(* IEC 61131-3 sources: teller/JD_Teller_LC2_V11/Class/Visu_Boxediter_MinMax, 1 file *)

(* ---- Visu_Boxediter_MinMax.st ---- *)
(*!
<Class
	Name               = "Visu_Boxediter_MinMax"
	Revision           = "1.2"
	RealtimeTask       = "false"
	CyclicTask         = "false"
	BackgroundTask     = "false"
	Sigmatek           = "false"
	OSInterface        = "false"
	HighPriority       = "false"
	Automatic          = "false"
	UpdateMode         = "Prescan"
	SharedCommandTable = "true"
	Objectsize         = "(750,1320)">
	<Channels>
		<Server Name="ClassSvr" Visualized="false" Initialize="false" WriteProtected="true" Retentive="false"/>
		<Server Name="s_BoxMogelijkopMachine" Visualized="true" Initialize="false" WriteProtected="false" Retentive="false"/>
		<Server Name="s_BoxType" Visualized="true" Initialize="false" WriteProtected="false" Retentive="false"/>
		<Server Name="s_Doosnaam" Visualized="true" Initialize="false" WriteProtected="true" Retentive="false"/>
		<Server Name="s_MaxLength" Visualized="true" Initialize="false" WriteProtected="false" Retentive="false"/>
		<Server Name="s_MaxWidth" Visualized="true" Initialize="false" WriteProtected="false" Retentive="false"/>
		<Server Name="s_Offset_Max" Visualized="true" Initialize="false" WriteProtected="false" Retentive="false"/>
		<Server Name="s_Offset_Min" Visualized="true" Initialize="false" WriteProtected="false" Retentive="false"/>
		<Server Name="s_Refresh_Values" Visualized="false" Initialize="false" WriteProtected="false" Retentive="false"/>
		<Server Name="s_T_Max" Visualized="true" Initialize="false" WriteProtected="false" Retentive="false"/>
		<Server Name="s_T_Min" Visualized="true" Initialize="false" WriteProtected="false" Retentive="false"/>
		<Server Name="s_U_Max" Visualized="true" Initialize="false" WriteProtected="false" Retentive="false"/>
		<Server Name="s_U_Min" Visualized="true" Initialize="false" WriteProtected="false" Retentive="false"/>
		<Server Name="s_V_Max" Visualized="true" Initialize="false" WriteProtected="false" Retentive="false"/>
		<Server Name="s_V_Min" Visualized="true" Initialize="false" WriteProtected="false" Retentive="false"/>
		<Server Name="s_W_Max" Visualized="true" Initialize="false" WriteProtected="false" Retentive="false"/>
		<Server Name="s_W_Min" Visualized="true" Initialize="false" WriteProtected="false" Retentive="false"/>
		<Server Name="s_X_Max" Visualized="true" Initialize="false" WriteProtected="false" Retentive="false"/>
		<Server Name="s_X_Min" Visualized="true" Initialize="false" WriteProtected="false" Retentive="false"/>
		<Server Name="s_Y_Max" Visualized="true" Initialize="false" WriteProtected="false" Retentive="false"/>
		<Server Name="s_Y_Min" Visualized="true" Initialize="false" WriteProtected="false" Retentive="false"/>
		<Server Name="s_Z_Max" Visualized="true" Initialize="false" WriteProtected="false" Retentive="false"/>
		<Server Name="s_Z_Min" Visualized="true" Initialize="false" WriteProtected="false" Retentive="false"/>
		<Client Name="c_Boxtype" Required="false" Internal="false"/>
		<Client Name="c_DoosData" Required="true" Internal="false"/>
		<Client Name="c_Refresh_Values" Required="true" Internal="false"/>
	</Channels>
	<RevDoku>
		<Owner Company="JD" Author="J van Diggelen"/>
		<Dokumentation Revision="1.2" Date="2014-04-29" Author="J van Diggelen" Company="JD" Description="doos 14 toegevoegd"/>
		<Dokumentation Revision="1.1" Date="2013-09-21" Author="J van Diggelen" Company="JD" Description="input warning opgelost"/>
		<Dokumentation Revision="1.0" Date="2011-12-06" Author="J van Diggelen" Company="JD" Description="De Visuwaarde van de Service settings van de boxeditor"/>
	</RevDoku>
</Class>
*)
Visu_Boxediter_MinMax : CLASS
  //Servers:
	ClassSvr 	: SvrChCmd_DINT;
	s_Doosnaam 	: SvrCh_tDoosnaam;
	s_BoxType 	: SvrCh_DINT;
	s_BoxMogelijkopMachine 	: SvrCh_DINT;
	s_MaxLength 	: SvrCh_DINT;
	s_MaxWidth 	: SvrCh_DINT;
	s_T_Max 	: SvrCh_DINT;
	s_T_Min 	: SvrCh_DINT;
	s_U_Max 	: SvrCh_DINT;
	s_U_Min 	: SvrCh_DINT;
	s_V_Max 	: SvrCh_DINT;
	s_V_Min 	: SvrCh_DINT;
	s_W_Max 	: SvrCh_DINT;
	s_W_Min 	: SvrCh_DINT;
	s_X_Max 	: SvrCh_DINT;
	s_X_Min 	: SvrCh_DINT;
	s_Y_Max 	: SvrCh_DINT;
	s_Y_Min 	: SvrCh_DINT;
	s_Z_Max 	: SvrCh_DINT;
	s_Z_Min 	: SvrCh_DINT;
	s_Offset_Max 	: SvrCh_DINT;
	s_Offset_Min 	: SvrCh_DINT;
	s_Refresh_Values 	: SvrCh_DINT;
  //Clients:
	c_DoosData 	: CltChCmd_RAMex;
	c_Boxtype 	: CltCh_DINT;
	c_Refresh_Values 	: CltCh_DINT;
  //Variables:
		DoosData 	: ^tDoosParameters;
  //Functions:

	FUNCTION VIRTUAL GLOBAL Init;

	FUNCTION VIRTUAL GLOBAL Background
		VAR_INPUT
			EAX 	: UDINT;
		END_VAR
		VAR_OUTPUT
			state (EAX) 	: UDINT;
		END_VAR;

	FUNCTION VIRTUAL GLOBAL s_BoxType::Write
		VAR_INPUT
			input (EAX) 	: DINT;
		END_VAR
		VAR_OUTPUT
			result (EAX) 	: DINT;
		END_VAR;

	FUNCTION VIRTUAL GLOBAL s_BoxMogelijkopMachine::Write
		VAR_INPUT
			input (EAX) 	: DINT;
		END_VAR
		VAR_OUTPUT
			result (EAX) 	: DINT;
		END_VAR;

	FUNCTION VIRTUAL GLOBAL s_MaxLength::Write
		VAR_INPUT
			input (EAX) 	: DINT;
		END_VAR
		VAR_OUTPUT
			result (EAX) 	: DINT;
		END_VAR;

	FUNCTION VIRTUAL GLOBAL s_MaxWidth::Write
		VAR_INPUT
			input (EAX) 	: DINT;
		END_VAR
		VAR_OUTPUT
			result (EAX) 	: DINT;
		END_VAR;

	FUNCTION VIRTUAL GLOBAL s_T_Max::Write
		VAR_INPUT
			input (EAX) 	: DINT;
		END_VAR
		VAR_OUTPUT
			result (EAX) 	: DINT;
		END_VAR;

	FUNCTION VIRTUAL GLOBAL s_T_Min::Write
		VAR_INPUT
			input (EAX) 	: DINT;
		END_VAR
		VAR_OUTPUT
			result (EAX) 	: DINT;
		END_VAR;

	FUNCTION VIRTUAL GLOBAL s_U_Max::Write
		VAR_INPUT
			input (EAX) 	: DINT;
		END_VAR
		VAR_OUTPUT
			result (EAX) 	: DINT;
		END_VAR;

	FUNCTION VIRTUAL GLOBAL s_U_Min::Write
		VAR_INPUT
			input (EAX) 	: DINT;
		END_VAR
		VAR_OUTPUT
			result (EAX) 	: DINT;
		END_VAR;

	FUNCTION VIRTUAL GLOBAL s_V_Max::Write
		VAR_INPUT
			input (EAX) 	: DINT;
		END_VAR
		VAR_OUTPUT
			result (EAX) 	: DINT;
		END_VAR;

	FUNCTION VIRTUAL GLOBAL s_V_Min::Write
		VAR_INPUT
			input (EAX) 	: DINT;
		END_VAR
		VAR_OUTPUT
			result (EAX) 	: DINT;
		END_VAR;

	FUNCTION VIRTUAL GLOBAL s_W_Max::Write
		VAR_INPUT
			input (EAX) 	: DINT;
		END_VAR
		VAR_OUTPUT
			result (EAX) 	: DINT;
		END_VAR;

	FUNCTION VIRTUAL GLOBAL s_W_Min::Write
		VAR_INPUT
			input (EAX) 	: DINT;
		END_VAR
		VAR_OUTPUT
			result (EAX) 	: DINT;
		END_VAR;

	FUNCTION VIRTUAL GLOBAL s_X_Max::Write
		VAR_INPUT
			input (EAX) 	: DINT;
		END_VAR
		VAR_OUTPUT
			result (EAX) 	: DINT;
		END_VAR;

	FUNCTION VIRTUAL GLOBAL s_X_Min::Write
		VAR_INPUT
			input (EAX) 	: DINT;
		END_VAR
		VAR_OUTPUT
			result (EAX) 	: DINT;
		END_VAR;

	FUNCTION VIRTUAL GLOBAL s_Y_Max::Write
		VAR_INPUT
			input (EAX) 	: DINT;
		END_VAR
		VAR_OUTPUT
			result (EAX) 	: DINT;
		END_VAR;

	FUNCTION VIRTUAL GLOBAL s_Y_Min::Write
		VAR_INPUT
			input (EAX) 	: DINT;
		END_VAR
		VAR_OUTPUT
			result (EAX) 	: DINT;
		END_VAR;

	FUNCTION VIRTUAL GLOBAL s_Z_Max::Write
		VAR_INPUT
			input (EAX) 	: DINT;
		END_VAR
		VAR_OUTPUT
			result (EAX) 	: DINT;
		END_VAR;

	FUNCTION VIRTUAL GLOBAL s_Z_Min::Write
		VAR_INPUT
			input (EAX) 	: DINT;
		END_VAR
		VAR_OUTPUT
			result (EAX) 	: DINT;
		END_VAR;

	FUNCTION VIRTUAL GLOBAL s_Offset_Max::Write
		VAR_INPUT
			input (EAX) 	: DINT;
		END_VAR
		VAR_OUTPUT
			result (EAX) 	: DINT;
		END_VAR;

	FUNCTION VIRTUAL GLOBAL s_Offset_Min::Write
		VAR_INPUT
			input (EAX) 	: DINT;
		END_VAR
		VAR_OUTPUT
			result (EAX) 	: DINT;
		END_VAR;

	FUNCTION VIRTUAL GLOBAL s_Refresh_Values::Write
		VAR_INPUT
			input (EAX) 	: DINT;
		END_VAR
		VAR_OUTPUT
			result (EAX) 	: DINT;
		END_VAR;
  //Tables:
	FUNCTION @STD
		VAR_OUTPUT
			ret_code	: CONFSTATES;
		END_VAR;
	FUNCTION GLOBAL TAB @CT_;
END_CLASS;

#pragma usingLtd RAMex

//Er is in de pointer variabele doosdata een array structuur gemaakt om bij elk type doos de minimale en maximale
//waardes in een service scherm te veranderen.

FUNCTION VIRTUAL GLOBAL Visu_Boxediter_MinMax::Init

  if c_DoosData.GetSize() <> sizeof(tDoosParameters) then
     c_DoosData.SetSize(udSize:=sizeof(tDoosParameters));
  end_if;

  if _FirstScan = 1 then

     DoosData := (c_DoosData.GetDataPtr())$^tDoosParameters;
     s_BoxType := c_Boxtype;
     s_BoxType.Write(s_BoxType);

  end_if;

END_FUNCTION

FUNCTION VIRTUAL GLOBAL Visu_Boxediter_MinMax::Background
	VAR_INPUT
		EAX 	: UDINT;
	END_VAR
	VAR_OUTPUT
		state (EAX) 	: UDINT;
	END_VAR

	state := READY;

END_FUNCTION

FUNCTION VIRTUAL GLOBAL Visu_Boxediter_MinMax::s_BoxType::Write
	VAR_INPUT
		input (EAX) 	: DINT;
	END_VAR
	VAR_OUTPUT
		result (EAX) 	: DINT;
	END_VAR

	s_BoxType := input;

  // doostype moet tussen 1 en 14 liggen
  if    s_BoxType <1 then
        s_BoxType :=1;
  elsif s_BoxType >14 then
        s_BoxType :=14;
  end_if;

 	result := s_BoxType;

  //Doostype
  if     s_BoxType = 1 then
         s_Doosnaam := Langsnaad;
  elsif  s_BoxType = 2 then
         s_Doosnaam := Driepunt;
  elsif  s_BoxType = 3 then
         s_Doosnaam := Driepunt_Vakverdeling;
  elsif  s_BoxType = 4 then
         s_Doosnaam := Vierpunt_Infold;
  elsif  s_BoxType = 5 then
         s_Doosnaam := Vierpunt_Outfold;
  elsif  s_BoxType = 6 then
         s_Doosnaam := Vierpunt_Deksel;
  elsif  s_BoxType = 7 then
         s_Doosnaam := Vierpunt_Dubbele_Wand;
  elsif  s_BoxType = 8 then
         s_Doosnaam := Zespunt_In_In;
  elsif  s_BoxType = 9 then
         s_Doosnaam := Zespunt_In_Out;
  elsif  s_BoxType = 10 then
         s_Doosnaam := Zespunt_In_In_Gespiegeld;
  elsif  s_BoxType = 11 then
         s_Doosnaam := Driepunt_Gespiegeld;
  elsif  s_BoxType = 12 then
         s_Doosnaam := Driepunt;
  elsif  s_BoxType = 13 then
         s_Doosnaam := Langsnaad2;
  elsif  s_BoxType = 14 then
         s_Doosnaam := Driepunt2;
  end_if;

  //Serverwaardes schrijven met variabelen voor type doos

  s_MaxLength := DoosData^.MinMax[s_BoxType].Max_Invoer_Lengte;
  s_MaxWidth  := DoosData^.MinMax[s_BoxType].Max_Invoer_Breedte;
  s_BoxMogelijkopMachine := DoosData^.MinMax[s_BoxType].BoxMogelijk;
  s_T_Max     := DoosData^.MinMax[s_BoxType].T_Max;
  s_T_Min     := DoosData^.MinMax[s_BoxType].T_Min;
  s_U_Max     := DoosData^.MinMax[s_BoxType].U_Max;
  s_U_Min     := DoosData^.MinMax[s_BoxType].U_Min;
  s_V_Min     := DoosData^.MinMax[s_BoxType].V_Min;
  s_V_Max     := DoosData^.MinMax[s_BoxType].V_Max;
  s_W_Max     := DoosData^.MinMax[s_BoxType].W_Max;
  s_W_Min     := DoosData^.MinMax[s_BoxType].W_Min;
  s_X_Max     := DoosData^.MinMax[s_BoxType].X_Max;
  s_X_Min     := DoosData^.MinMax[s_BoxType].X_Min;
  s_Y_Max     := DoosData^.MinMax[s_BoxType].Y_Max;
  s_Y_Min     := DoosData^.MinMax[s_BoxType].Y_Min;
  s_Z_Max     := DoosData^.MinMax[s_BoxType].Z_Max;
  s_Z_Min     := DoosData^.MinMax[s_BoxType].Z_Min;
  s_Offset_Max:= DoosData^.MinMax[s_BoxType].Offset_Max;
  s_Offset_Min:= DoosData^.MinMax[s_BoxType].Offset_Min;

END_FUNCTION

FUNCTION VIRTUAL GLOBAL Visu_Boxediter_MinMax::s_BoxMogelijkopMachine::Write
	VAR_INPUT
		input (EAX) 	: DINT;
	END_VAR
	VAR_OUTPUT
		result (EAX) 	: DINT;
	END_VAR

  s_BoxMogelijkopMachine := input;
  DoosData^.MinMax[s_BoxType].BoxMogelijk := to_bool(s_BoxMogelijkopMachine);
  c_Refresh_Values.Write(input:=1);
  result := s_BoxMogelijkopMachine;

END_FUNCTION

FUNCTION VIRTUAL GLOBAL Visu_Boxediter_MinMax::s_MaxLength::Write
	VAR_INPUT
		input (EAX) 	: DINT;
	END_VAR
	VAR_OUTPUT
		result (EAX) 	: DINT;
	END_VAR

	s_MaxLength := input;
  DoosData^.MinMax[s_BoxType].Max_Invoer_Lengte := s_MaxLength;
  c_Refresh_Values.Write(input:=1);
 	result := s_MaxLength;

END_FUNCTION

FUNCTION VIRTUAL GLOBAL Visu_Boxediter_MinMax::s_MaxWidth::Write
	VAR_INPUT
		input (EAX) 	: DINT;
	END_VAR
	VAR_OUTPUT
		result (EAX) 	: DINT;
	END_VAR

	s_MaxWidth := input;
  DoosData^.MinMax[s_BoxType].Max_Invoer_Breedte := s_MaxWidth;
  c_Refresh_Values.Write(input:=1);
 	result := s_MaxWidth;

END_FUNCTION

FUNCTION VIRTUAL GLOBAL Visu_Boxediter_MinMax::s_T_Max::Write
	VAR_INPUT
		input (EAX) 	: DINT;
	END_VAR
	VAR_OUTPUT
		result (EAX) 	: DINT;
	END_VAR

	s_T_Max := input;
  DoosData^.MinMax[s_BoxType].T_Max:= s_T_Max;
  c_Refresh_Values.Write(input:=1);
 	result := s_T_Max;

END_FUNCTION

FUNCTION VIRTUAL GLOBAL Visu_Boxediter_MinMax::s_T_Min::Write
	VAR_INPUT
		input (EAX) 	: DINT;
	END_VAR
	VAR_OUTPUT
		result (EAX) 	: DINT;
	END_VAR

	s_T_Min := input;
  DoosData^.MinMax[s_BoxType].T_Min:= s_T_Min;
  c_Refresh_Values.Write(input:=1);
 	result := s_T_Min;

END_FUNCTION

FUNCTION VIRTUAL GLOBAL Visu_Boxediter_MinMax::s_U_Max::Write
	VAR_INPUT
		input (EAX) 	: DINT;
	END_VAR
	VAR_OUTPUT
		result (EAX) 	: DINT;
	END_VAR

	s_U_Max := input;
  DoosData^.MinMax[s_BoxType].U_Max:=s_U_Max;
  c_Refresh_Values.Write(input:=1);
 	result := s_U_Max;

END_FUNCTION

FUNCTION VIRTUAL GLOBAL Visu_Boxediter_MinMax::s_U_Min::Write
	VAR_INPUT
		input (EAX) 	: DINT;
	END_VAR
	VAR_OUTPUT
		result (EAX) 	: DINT;
	END_VAR

	s_U_Min := input;
  DoosData^.MinMax[s_BoxType].U_Min:= s_U_Min;
  c_Refresh_Values.Write(input:=1);
 	result := s_U_Min;

END_FUNCTION

FUNCTION VIRTUAL GLOBAL Visu_Boxediter_MinMax::s_V_Max::Write
	VAR_INPUT
		input (EAX) 	: DINT;
	END_VAR
	VAR_OUTPUT
		result (EAX) 	: DINT;
	END_VAR

	s_V_Max := input;
  DoosData^.MinMax[s_BoxType].V_Max:=s_V_Max;
  c_Refresh_Values.Write(input:=1);
 	result := s_V_Max;

END_FUNCTION

FUNCTION VIRTUAL GLOBAL Visu_Boxediter_MinMax::s_V_Min::Write
	VAR_INPUT
		input (EAX) 	: DINT;
	END_VAR
	VAR_OUTPUT
		result (EAX) 	: DINT;
	END_VAR

	s_V_Min := input;
  DoosData^.MinMax[s_BoxType].V_Min:=s_V_Min;
  c_Refresh_Values.Write(input:=1);
 	result := s_V_Min;

END_FUNCTION

FUNCTION VIRTUAL GLOBAL Visu_Boxediter_MinMax::s_W_Max::Write
	VAR_INPUT
		input (EAX) 	: DINT;
	END_VAR
	VAR_OUTPUT
		result (EAX) 	: DINT;
	END_VAR

	s_W_Max := input;
  DoosData^.MinMax[s_BoxType].W_Max:=s_W_Max;
  c_Refresh_Values.Write(input:=1);
 	result := s_W_Max;

END_FUNCTION

FUNCTION VIRTUAL GLOBAL Visu_Boxediter_MinMax::s_W_Min::Write
	VAR_INPUT
		input (EAX) 	: DINT;
	END_VAR
	VAR_OUTPUT
		result (EAX) 	: DINT;
	END_VAR

	s_W_Min := input;
  DoosData^.MinMax[s_BoxType].W_Min:=s_W_Min;
  c_Refresh_Values.Write(input:=1);
 	result := s_W_Min;

END_FUNCTION

FUNCTION VIRTUAL GLOBAL Visu_Boxediter_MinMax::s_X_Max::Write
	VAR_INPUT
		input (EAX) 	: DINT;
	END_VAR
	VAR_OUTPUT
		result (EAX) 	: DINT;
	END_VAR

	s_X_Max := input;
  DoosData^.MinMax[s_BoxType].X_Max:=s_X_Max;
  c_Refresh_Values.Write(input:=1);
 	result := s_X_Max;

END_FUNCTION

FUNCTION VIRTUAL GLOBAL Visu_Boxediter_MinMax::s_X_Min::Write
	VAR_INPUT
		input (EAX) 	: DINT;
	END_VAR
	VAR_OUTPUT
		result (EAX) 	: DINT;
	END_VAR

	s_X_Min := input;
  DoosData^.MinMax[s_BoxType].X_Min:=s_X_Min;
  c_Refresh_Values.Write(input:=1);
 	result := s_X_Min;

END_FUNCTION

FUNCTION VIRTUAL GLOBAL Visu_Boxediter_MinMax::s_Y_Max::Write
	VAR_INPUT
		input (EAX) 	: DINT;
	END_VAR
	VAR_OUTPUT
		result (EAX) 	: DINT;
	END_VAR

	s_Y_Max := input;
  DoosData^.MinMax[s_BoxType].Y_Max:=s_Y_Max;
  c_Refresh_Values.Write(input:=1);
 	result := s_Y_Max;

END_FUNCTION

FUNCTION VIRTUAL GLOBAL Visu_Boxediter_MinMax::s_Y_Min::Write
	VAR_INPUT
		input (EAX) 	: DINT;
	END_VAR
	VAR_OUTPUT
		result (EAX) 	: DINT;
	END_VAR

	s_Y_Min := input;
  DoosData^.MinMax[s_BoxType].Y_Min:= s_Y_Min;
  c_Refresh_Values.Write(input:=1);
 	result := s_Y_Min;

END_FUNCTION

FUNCTION VIRTUAL GLOBAL Visu_Boxediter_MinMax::s_Z_Max::Write
	VAR_INPUT
		input (EAX) 	: DINT;
	END_VAR
	VAR_OUTPUT
		result (EAX) 	: DINT;
	END_VAR

	s_Z_Max := input;
  DoosData^.MinMax[s_BoxType].Z_Max:= s_Z_Max;
  c_Refresh_Values.Write(input:=1);
 	result := s_Z_Max;

END_FUNCTION

FUNCTION VIRTUAL GLOBAL Visu_Boxediter_MinMax::s_Z_Min::Write
	VAR_INPUT
		input (EAX) 	: DINT;
	END_VAR
	VAR_OUTPUT
		result (EAX) 	: DINT;
	END_VAR

	s_Z_Min := input;
  DoosData^.MinMax[s_BoxType].Z_Min:= s_Z_Min;
  c_Refresh_Values.Write(input:=1);
 	result := s_Z_Min;

END_FUNCTION

FUNCTION VIRTUAL GLOBAL Visu_Boxediter_MinMax::s_Offset_Max::Write
	VAR_INPUT
		input (EAX) 	: DINT;
	END_VAR
	VAR_OUTPUT
		result (EAX) 	: DINT;
	END_VAR

	s_Offset_Max := input;
  DoosData^.MinMax[s_BoxType].Offset_Max:= s_Offset_Max;
  c_Refresh_Values.Write(input:=1);
 	result := s_Offset_Max;

END_FUNCTION

FUNCTION VIRTUAL GLOBAL Visu_Boxediter_MinMax::s_Offset_Min::Write
	VAR_INPUT
		input (EAX) 	: DINT;
	END_VAR
	VAR_OUTPUT
		result (EAX) 	: DINT;
	END_VAR

	s_Offset_Min := input;
  DoosData^.MinMax[s_BoxType].Offset_Min:= s_Offset_Min;
  c_Refresh_Values.Write(input:=1);
 	result := s_Offset_Min;

END_FUNCTION

FUNCTION VIRTUAL GLOBAL Visu_Boxediter_MinMax::s_Refresh_Values::Write

	VAR_INPUT
		input (EAX) 	: DINT;
	END_VAR
	VAR_OUTPUT
		result (EAX) 	: DINT;
	END_VAR

	s_Refresh_Values := input;
  s_Refresh_Values := 0;
  s_BoxType.Write(s_BoxType);
 	result := s_Refresh_Values;

END_FUNCTION
